KUKA KRL data list: TEST_ToolMeasure.dat

&ACCESS RVO
&REL 58
&PARAM DISKPATH = KRC:\R1\Program\Test\ToolMagazine
DEFDAT  TEST_ToolMeasure

DECL CONST INT iSafetyStop=11
DECL CONST INT iMeasureStop=12

DECL POS xSpindle
DECL REAL rToolLength=-1.00000

DECL CONST REAL rToolLengthMin=120.000
DECL CONST REAL rToolLengthMax=230.000
DECL CONST REAL rMeasureOffset=10.0000

DECL CONST POS xSensor={X 725.700,Y -70.5000,Z 63.6000,A 0.0,B 0.0,C 0.0}
DECL CONST FRAME fAboveSensor={X 0.0,Y 0.0,Z 300.000,A 0.0,B 0.0,C 0.0}
DECL CONST FRAME fMeasureOffset={X 0.0,Y 0.0,Z 10.0000,A 0.0,B 0.0,C 0.0}

DECL CONST FRAME fMeasureStart={X 0.0,Y 0.0,Z 250.000,A 0.0,B 0.0,C 0.0}
DECL CONST FRAME fMeasureEnd={X 0.0,Y 0.0,Z 100.000,A 0.0,B 0.0,C 0.0}

DECL CONST FRAME fToolMeasured={X 0.0,Y 0.0,Z 15.0000,A 0.0,B 0.0,C 0.0}

ENDDAT
